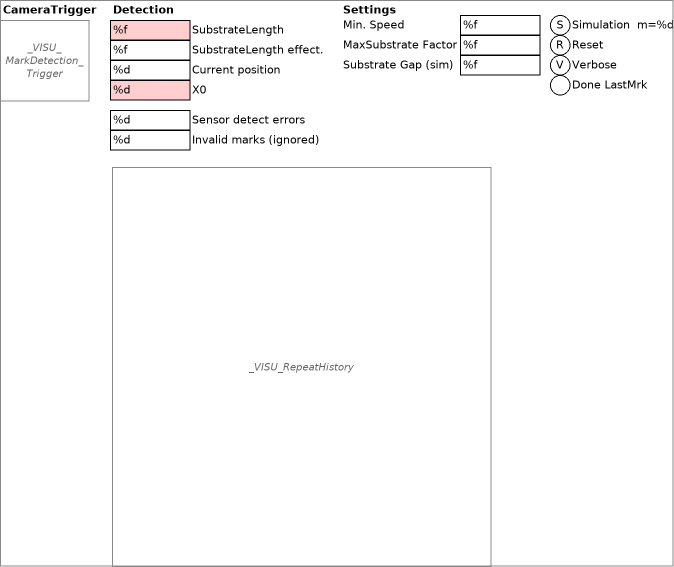
VISUALIZATION _VISU_MarkDetection  // 674x567
VAR_IN_OUT
	mInst: FB_MarkDetection;
END_VAR
    Ellipse (550,35 20x20), "R", tooltip "Reset"
        tap mInst.bManualReset
    Frame (0,20 89x81)
        shows _VISU_MarkDetection_Trigger(mInst := mInst)
    Rectangle (0,0 100x20), "CameraTrigger"
    Rectangle (110,20 80x20), "%f", text variable: mInst._fSubstrateLength, colour toggle: mInst._fSubstrateLength > 0
    Rectangle (189,20 140x20), "SubstrateLength"
    Rectangle (110,40 80x20), "%f", text variable: mInst._fSubstrateLengthEffective
    Rectangle (189,40 140x20), "SubstrateLength effect."
    Rectangle (110,80 80x20), "%d", text variable: mInst._nX0, colour toggle: mInst._bValid
    Rectangle (189,80 140x20), "X0"
    Rectangle (110,60 80x20), "%d", text variable: mInst.nCurrentPos
    Rectangle (189,60 140x20), "Current position"
    Ellipse (550,15 20x20), "S", tooltip "Simulation"
        toggle mInst._bSimEnable
    Rectangle (569,15 100x20), "Simulation"
    Ellipse (550,75 20x20)
        toggle mInst.bR_TerminateLast
    Rectangle (569,75 100x20), "Done LastMrk"
    Rectangle (569,35 100x20), "Reset"
    Ellipse (550,55 20x20), "V", tooltip "Verbose"
        toggle mInst._bVerbose
    Rectangle (569,55 100x20), "Verbose"
    Rectangle (460,15 80x20), "%f", text variable: mInst.fC_MinimalSpeed, input disabled if: TRUE
    Rectangle (340,15 120x20), "Min. Speed"
    Rectangle (460,35 80x20), "%f", text variable: mInst.fC_MaxSubstrateFactor, input disabled if: TRUE
    Rectangle (340,35 120x20), "MaxSubstrate Factor"
    Rectangle (460,55 80x20), "%f", text variable: mInst._fSubstrateGap, invisible if: NOT mInst._bSimEnable
        OnMouseClick: write the text variable via Default
    Rectangle (340,55 120x20), "Substrate Gap (sim)", invisible if: NOT mInst._bSimEnable
    Rectangle (110,0 100x20), "Detection"
    Rectangle (340,0 100x20), "Settings"
    RoundedRectangle (110,110 80x20), "%d", text variable: mInst.nCtrSensorDetectError, colour toggle: mInst.nCtrSensorDetectError > 0
    Rectangle (189,110 140x20), "Sensor detect errors"
    RoundedRectangle (110,130 80x20), "%d", text variable: mInst.nCtrIgnoredMarks, colour toggle: mInst.nCtrIgnoredMarks > 0
    Rectangle (189,130 140x20), "Invalid marks (ignored)"
    TabControl (112,167 379x400)
        shows _VISU_RepeatHistory(mInst := mInst)
        shows _VISU_MarkHistory(mInst := mInst)
        [0]: TabTitle=Repeat History
        [1]: TabTitle=Mark History
    Rectangle (634,15 40x20), "m=%d", tooltip "simulation mode", text variable: mInst._nSimMode
        OnMouseClick: write the text variable via Default
END_VISUALIZATION

(* stored: Version 1.1.0.1, ProductVersion 3.1.4024.11
   Visu _VISU_MarkDetection: Id {2a376e8e-8ddc-405b-aef1-8180a4580dbe} *)
